// TIA Portal V19 export
TYPE "udt_BimanualSts"
// stored: Access Published, IsFailsafeCompliant true
   STRUCT
      SafeMotion : Bool;
      Enable : Bool;
   END_STRUCT;
END_TYPE
